PROGRAM MAIN
VAR
	fb_led_Show: FB_LedShow;
	btn_reset: BOOL;
	CPMU_PLC_Reset: PLC_Reset;
	d_state: DINT;
	CPMU_PLC_Start: PLC_Start;
	powerStatus:BOOL;

(*TwinSAFE*)
	Safe_run AT%Q*:BOOL;
	Err_Ack AT %Q*:BOOL;
	Estop_RunAndRestart AT %Q*:BOOL;
	AX5805_Error_Ack AT %Q*:BOOL;
	Led_Run  AT %Q*:BOOL;
	Led_Error  AT %Q*:BOOL;

	FB_ERROR AT%I*:BOOL;
	COM_ERROR AT%I*:BOOL;
	//OUT_ERROR AT%I*:BOOL;
	Estop_Out AT%I*:BOOL;

	SafeStatus:INT;
	SafePLCRunOK: BOOL;
	fb_ton: TON;
	fb_ton2: TON;
	fb_ton3: TON;
	fb_ton1: TON;
	fb_ton0: TON;
(*IO*)
	el1808_D1  AT%I* :ARRAY[1..4] OF BOOL;
	el1008 AT%I*:BOOL;
	EStopTrig:BOOL;
(*setAxisPosition*)
	SetAxisPosState: INT;
	FB_Set_AxisPosition:FB_SetAxisPosition;
	fb_ton4: TON;
	fb_ton5: TON;
	fb_ton6: TON;
	SetAxisPositionDone: BOOL;

	i: INT;
	j: INT;

(****RS232***)
	fbEL6001	: FB_SerialCom;
	
	moveDonePhaseShifter: BOOL;


(*Torque*)
	Torque_PS AT%I*:INT;
(**)
	btn_setAxisPosition: BOOL;
	ValueSet_PhaseShifterLin:LREAL;
(**)
	RestartTC: TC_Restart;
	
(*recipe*)
	RecipeINT:INT;
	RecipeBOOL:BOOL;
	RecipeManCommands: RecipeManCommands;
	SaveParameter : BOOL;  //保存文件
	LoadParameter : BOOL;  //读取文件
	Save_R_TRIG   : R_TRIG;
	Read_R_TRIG   : R_TRIG;
	loadparameterStatus: INT;
	RecipeBOOL2:BOOL;
	ReturnDwordLoad: DWORD;
	InsertionDeviceName:STRING;
(*UserMode*)
	pbUserMode: BOOL:=TRUE;
	EL1904 AT%I* :ARRAY[1..24] OF BOOL;
	setAxisPositionEnable: BOOL;
	state_loadParameters: INT;
	state_setLEPosBias: INT;
	//
	PositionBiasSet:BOOL;
	MC_SetLEPosBias_PhaseShifter:MC_WriteParameter;
	PositionBias_PhaseShifter: LREAL:=10.1;
	LoadLEPB_R_TRIG: R_TRIG;
	PositionBiasTON: TON;
	
	//
	OPC_TEST_Bi:BOOL:=TRUE; (*~ (OPC:1:available for OPC Clients) *)
	OPC_TEST_Bi2:BOOL;(*~ (OPC:1:available for OPC Clients) *)
	//
	HasTemperatureSensorOrNot:BOOL;//Only IVU or CPMU
	(*Sensor Reading*)
	Sensor_Reading_1 AT %I*:ARRAY[0..3] OF BYTE;
	Sensor_Reading_2 AT %I*:ARRAY[0..3] OF BYTE;
	Sensor_Reading_3 AT %I*:ARRAY[0..3] OF BYTE;
	Sensor_Reading_4 AT %I*:ARRAY[0..3] OF BYTE;
	Sensor_Reading_5 AT %I*:ARRAY[0..3] OF BYTE;
	Sensor_Reading_6 AT %I*:ARRAY[0..3] OF BYTE;
	Sensor_Reading_7 AT %I*:ARRAY[0..3] OF BYTE;
	Sensor_Reading_8 AT %I*:ARRAY[0..3] OF BYTE;
	Sensor_Reading_DpState AT %I*:USINT;
	Sensor_Reading_ExtDiagFlag AT %I*:BOOL;
	TemperatureSensors_1:LREAL;
	TemperatureSensors_2:LREAL;
	TemperatureSensors_3:LREAL;
	TemperatureSensors_4:LREAL;
	TemperatureSensors_5:LREAL;
	TemperatureSensors_6:LREAL;
	TemperatureSensors_7:LREAL;
	TemperatureSensors_8:LREAL;
	dut_sensor_datas_1:DUT_SENSOR_DATAS_1;
	dut_sensor_datas_2:DUT_SENSOR_DATAS_2;
	dut_sensor_datas_3:DUT_SENSOR_DATAS_3;
	dut_sensor_datas_4:DUT_SENSOR_DATAS_4;
	dut_sensor_datas_5:DUT_SENSOR_DATAS_5;
	dut_sensor_datas_6:DUT_SENSOR_DATAS_6;
	dut_sensor_datas_7:DUT_SENSOR_DATAS_7;
	dut_sensor_datas_8:DUT_SENSOR_DATAS_8;
	//
	temperature_gradient_2_To_1:LREAL;
	temperature_gradient_3_To_2:LREAL;
	temperature_gradient_5_To_4:LREAL;
	temperature_gradient_6_To_5:LREAL;
	temperature_gradient_max:LREAL;
	//
	temperature_average:LREAL;
	A_SetLinearEncoderPositionBias_Enable: BOOL;
	
		//
	temperatureStatus:INT;//0：有传感器度数错误；1:常温；2:低温；3:常温和低温中间态
	CryogenicTemperatureThreshold:LREAL:=80;//80K以下归划分为低温
	RoomTemperatureThreshold:LREAL:=293;//293K以上划分为常温
	//CPMU cryogenix ON/FF
	CryogenicCompensationOn:BOOL;
	CryogenicCompensationConditionsReady:BOOL;
	CryogenicCompensation_LeftTop:LREAL;
	CryogenicCompensation_RightTop:LREAL;
	CryogenicCompensation_LeftBottom:LREAL;
	CryogenicCompensation_RightBottom:LREAL;
	CryogenicCompensationDone: BOOL;
	
(**)
	bDriveDiagMessageAndNumber  : BOOL;
	m_GetDriveStatusState:INT;
	GetDriveStatusStateDone:BOOL;
	GetDriveStatusStateError:BOOL;
	GetDriveStatusTON: TON;
	//	
	fb_SoEReadDiagMessage_PhaseShifter: FB_SoEReadDiagMessage;
	DriveDiagMessage_PhaseShifter:STRING;
	//
	FB_SoEReadDiagNumber_PhaseShifter: FB_SoEReadDiagNumber;
	DriveDiagNumber_PhaseShifter:UDINT;
	bReloadDriveDiagMessageAndNumber: BOOL;
	
	(*load IOC*)
	bExe_load_Prog: BOOL;
	NT_StartProcess_Load: NT_StartProcess;
	Exe_load_step: UINT;
	R_TRIG_ExeLoad: R_TRIG;
	Exe_Load_Done:BOOL;
	(*kill IOC*)
	bExe_Kill_Prog: BOOL;
	NT_StartProcess_Kill: NT_StartProcess;
	Exe_kill_step: UINT;
	R_TRIG_Exekill: R_TRIG;
	Exe_Kill_Done:BOOL;

	KS_RightBottom_Near_Contact2: BOOL;
	
	//
	//more parameters get:gear;feedback2 direction 
	//
	//GetMoreDriveStatus_FunctionON:BOOL:=TRUE;
	GetDriveStatusTON2: TON;
	//GearNumerator,st182
	st_p182_PhaseShifter:ST_P182;
	FB_SoERead_GearNumerator_PhaseShifter: FB_SoERead;
	GearNumeratorGet_PhaseShifter:UDINT;
	GearNumeratorConfigured_PhaseShifter:UDINT;
	//GearDenominator,st183
	st_p183_PhaseShifter:ST_P183;
	FB_SoERead_GearDenominator_PhaseShifter: FB_SoERead;
	GearDenominatorGet_PhaseShifter:UDINT;
	GearDenominatorConfigured_PhaseShifter:UDINT;
	//Feedback2direction,st180
	st_p180_PhaseShifter:ST_P180;
	FB_SoERead_Feedback2direction_PhaseShifter: FB_SoERead;
	Feedback2directionGet_PhaseShifter:UINT;
	Feedback2directionConfigured_PhaseShifter:UINT;
	//
	//RestartDrivers
		(*重启驱动器*)
	btn_RestartDriversAll:BOOL;
	btn_RestartDriver1:BOOL;
	btn_RestartDriver2:BOOL;
	btn_RestartDriver3:BOOL;
	btn_RestartDriver4:BOOL;
	btn_RestartDriver5:BOOL;
	btn_RestartDriver6:BOOL;
	btn_RestartDriver7:BOOL;
	btn_RestartDriver8:BOOL;
	Relay_EL2624 AT %Q*:ARRAY[0..7]OF  BOOL;
	RestartDriver_RTRIG:R_TRIG;
	RestartDriver_TON:TON;
	RestartDriver_Triggered:BOOL;
	RestartDriver_State:DINT;
	RestartDriver_Done:BOOL;
	
	//
	//	LEHeartBeatMonitorFunction
	//
	LEHeartBeatMonitorFunctionOn: BOOL;
	LEHeartBeatFirstScan:BOOL;
	LEHeartBeatDeadZone : LREAL := 0; 
	LEHeartBeatAlarmTime : TIME := T#0.1S;
	
    //Pos_LeftTopLin_Last : LREAL; 
	Velo_PhaseShifterLin_Last : LREAL; 
	Pos_PhaseShifterMotor_Initial : LREAL; 
    StableTimer_PhaseShifterLin : TON; 
    StableTime_PhaseShifterLin : TIME; 
    DeltaVelo_PhaseShifterLin : LREAL; 
	IsInitialPositionSet_PhaseShifter: BOOL;
	MotorPosChange_PhaseShifter: LREAL;
	Threshold_PhaseShifterMotorPos:LREAL:=0.1;
	Threshold_PhaseShifterMotorVelo:LREAL:=0.2;
	Alarm_PhaseShifterLin:BOOL;
	Alarm_PhaseShifterMotorPos:BOOL;
	Alarm_PhaseShifterMotorVelo:BOOL;
	
	(*setAxisPosition*)
	SetMotorAxisPosState: INT;
	FB_Set_MotorAxisPosition:FB_SetMotorAxisPosition;
	fb_ton4_2: TON;
	fb_ton5_2: TON;
	fb_ton6_2: TON;
	SetMotorAxisPositionDone: BOOL;
	
	btn_SetMotorAxisPosition: BOOL;
	MonitorMotorAndLEFunctionOn:BOOL:=TRUE;
	
	(*GetMotorTempture*)
	MotorTemperature AT %I*:ARRAY[0..1] OF UINT;
	MotorTemperature_PS:LREAL;
END_VAR

(*MaintenanceMode*)
IF MaintenanceMode THEN
	MaintenanceModeLed:=TRUE;
	RETURN;
ELSE
	MaintenanceModeLed:=FALSE;	
END_IF

(*加载Ricipe参数*)
A_InitRecipeParameters();
(*Restart TwinCAT*)
IF Global_Variables.m_restartTC THEN
(*首先关闭opcIocShell.exe*)	
	bExe_Kill_Prog:=TRUE;
	A_KillOpcIocShellExe();
(*重启TC*)
	IF Exe_Kill_Done THEN
		A_RestartTC();
	END_IF
END_IF
(*******InitAxisParameters*******)
A_InitAxisParameters();
(*******CheckLimitSwitch*******)
A_CheckLimitSwitch();
(*Check Kill Switch*)
A_CheckKillSwitch();
(*******PosDiff¼à¿Ø*******)
A_PosDiffDetectiion();
(*******³õÊ¼»¯SafePlc*******)
IF NOT simulation THEN
A_SafePlcStartInit();
END_IF
(************SetAxisPosition*********************)
IF  NOT USELinearEncoder AND setAxisPositionEnable AND btn_setAxisPosition THEN
	//IF NOT SerAxisPositionDone THEN
		FB_Set_AxisPosition.ValueSet_PhaseShifterLin:=ValueSet_PhaseShifterLin;
		A_SetAxisPosition();
	//END_IF
END_IF
(*******³Mode Select******)
IF SafePLCRunOK OR Simulation THEN
	UserMode();
END_IF
(*******Led Show******)
fb_led_Show();
(*******Check Power status******)
FB_Power(Check:=TRUE);
st_Power:=FB_Power.PowerState;
(*********RS232*********************)
BackgroundEL();
(*fbEL6001(TxBuffer:=TxBufferEL, RxBuffer:=RxBufferEL);*)

(*设置position bias*)
IF loadParametersDone AND (DriveStatus=1 OR simulation) THEN 
	A_SetLinearEncoderPositionBias();
END_IF
(*检查硬急停状态，包括安全限位、柜门急停、手持急停*)
A_CheckHardwareEmergencyStopStatus();
(*获取驱动器状态信息*)
IF NOT simulation THEN
	A_GetDriverStatus();
END_IF
(*IDControlReady*)
IF ((DriveStatus<>0 AND SafePLCRunOK) OR simulation) AND NOT Error THEN
	IDControlReady:=TRUE;
ELSE
	IDControlReady:=FALSE;
END_IF

(*IOC Start*)
//IF IDControlReady THEN
	bExe_load_Prog:=TRUE;
	A_LoadOpcIocShellExe();
//END_IF

(*检查光栅读数是否在范围内*)
A_CheckLinearEncoder();

(*RestartDrivers*)
A_RestartDrivers();

(*A_LEHeartBeatMonitor*)
IF LEHeartBeatMonitorFunctionOn THEN
	A_LEHeartBeatMonitor();
END_IF
(************SetMotorAxisPosition*********************)
//IDControl 1s after
fb_ton5_2.IN:=IDControlReady;
fb_ton5_2.PT:=T#1S;
fb_ton5_2();
IF fb_ton5_2.Q THEN
	btn_SetMotorAxisPosition:=TRUE;
END_IF
IF  USELinearEncoder AND btn_SetMotorAxisPosition THEN
	IF NOT SetMotorAxisPositionDone THEN
		FB_Set_MotorAxisPosition.ValueSet_PhaseShifterMotor:=Pos_PhaseShifterLin;
		A_SetMotorAxisPosition();
	END_IF
END_IF
(*A_MonitorMotorAndLE*)
IF MonitorMotorAndLEFunctionOn AND SetMotorAxisPositionDone THEN
	A_MonitorMotorAndLE();
END_IF
(*A_CheckMaxVelocity*)
A_CheckMaxVelocity();

ACTION A_CheckHardwareEmergencyStopStatus:
IF 	NOT KS_TopNear_Contact1 OR
	NOT KS_TopNear_Contact2 OR
	NOT KS_TopFar_Contact1 OR
	NOT KS_TopFar_Contact2 OR
	
(*E-STOP*)
	NOT KS_CabinetEmergency_contact1 OR
	NOT KS_CabinetEmergency_contact2 OR
	NOT KS_handEmergency1_Contact1 OR
	NOT KS_handEmergency1_Contact2 OR
	NOT KS_handEmergency2_Contact1 OR
	NOT KS_handEmergency2_Contact2 OR
	NOT KS_softEmergency2_Contact THEN
	Hardware_EmergencyStop:=FALSE;
ELSE
	Hardware_EmergencyStop:=TRUE;
END_IF
END_ACTION

ACTION A_CheckKillSwitch:
IF simulation THEN	
	KS_TopFar_Contact1:=TRUE;	
	KS_TopFar_Contact2:=TRUE;	
	KS_TopNear_Contact1:=TRUE;	
	KS_TopNear_Contact2:=TRUE;	
	KS_BottomFar_Contact1:=TRUE;	
	KS_BottomFar_Contact2:=TRUE;	
	KS_BottomNear_Contact1:=TRUE;	
	KS_BottomNear_Contact2:=TRUE;	
	(*E-STOP*)
	KS_CabinetEmergency_contact1:=TRUE;
	KS_CabinetEmergency_contact2:=TRUE;	
	KS_handEmergency1_Contact1:=TRUE;
	KS_handEmergency1_Contact2:=TRUE;
	KS_handEmergency2_Contact1:=TRUE;
	KS_handEmergency2_Contact2:=TRUE;
	
	KS_softEmergency2_Contact:=TRUE;

ELSE
	KS_TopFar_Contact1:=EL1904[1];//c1	
	KS_TopFar_Contact2:=EL1904[2];//c1	
	KS_TopNear_Contact1:=EL1904[3];//c1	
	KS_TopNear_Contact2:=EL1904[4];//c1	
	KS_BottomFar_Contact1:=EL1904[5];//c2	
	KS_BottomFar_Contact2:=EL1904[6];//c2	
	KS_BottomNear_Contact1:=EL1904[7];//c2	
	KS_BottomNear_Contact2:=EL1904[8];//c2
	
	
	(*E-STOP*)
	KS_CabinetEmergency_contact1:=EL1904[9];//c3
	KS_CabinetEmergency_contact2:=EL1904[10];//c3
	
	KS_handEmergency1_Contact1:=EL1904[11];//c3
	KS_handEmergency1_Contact2:=EL1904[12];//c3
	KS_handEmergency2_Contact1:=EL1904[13];//c4
	KS_handEmergency2_Contact2:=EL1904[14];//c4
	
	KS_softEmergency2_Contact:=EL1904[15];//c4
	//c4
	END_IF
END_ACTION

ACTION A_CheckLimitSwitch:
(*******1.´ÓIO»ñÈ¡ÏÞÎ»×´Ì¬******)
(**)
IF simulation THEN
	(**)
	LS_TopFar  :=TRUE;
	LS_TopNear :=TRUE;
	LS_BottomFar :=TRUE;
	LS_BottomNear  :=TRUE;
ELSE
	LS_TopFar  :=el1808_D1[1];
	LS_TopNear :=el1808_D1[2];
	LS_BottomFar :=el1808_D1[3];
	LS_BottomNear :=el1808_D1[4];

END_IF
(******2.TopÏÞÎ»»òÕßBottomÏÞÎ»ÓÐÒ»¸ö´¥·¢£¬È«¾Ö±äÁ¿¡£¸øMC_POWERÓÃÓÚ·½Ïò¿ØÖÆ£¬ÓÐÒ»¸öÏÞÎ»Îª´¥·¢ÎªFALSE£¬ÔòUnreach_LSÎªFALSE******)
//Unreach_LS_Far:=LS_TopFar AND LS_BottomFar;
//Unreach_LS_Near:=LS_TopNear AND LS_BottomNear;

Unreach_LS_Far:=LS_TopFar;
Unreach_LS_Near:=LS_TopNear;
END_ACTION

ACTION A_CheckLinearEncoder:
//LEProtectionPosition
min_UserLEProtectionGapPosition:=min_UserGapPositionNew-min_ThresholdGapSoft2LEProtection;//回程误差有0.1mm
max_UserLEProtectionGapPosition:=max_UserGapPositionNew+max_ThresholdGapSoft2LEProtection;

//如果没有使用光栅、或者光栅参数没设置好，则不检查光栅位置
IF NOT USELinearEncoder OR NOT PositionBiasDone THEN
	RETURN;
END_IF
IF Pos_PhaseShifterLin <=0 THEN
	ErrorID:=1101;
	Error:=TRUE;
	ErrorDescription:='Pos_PhaseShifterLin <=0';
	FB_PlcEmergencyStop();
	LED_Error:=TRUE;
END_IF
//

IF Pos_PhaseShifterLin >max_UserLEProtectionGapPosition THEN
	ErrorID:=1105;
	Error:=TRUE;
	ErrorDescription:='Pos_PhaseShifterLin >max_UserLEProtectionGapPosition';
	FB_PlcEmergencyStop();
	LED_Error:=TRUE;
END_IF

//
IF Pos_PhaseShifterLin <min_UserLEProtectionGapPosition THEN
	ErrorID:=1109;
	Error:=TRUE;
	ErrorDescription:='Pos_PhaseShifterLin <min_UserLEProtectionGapPosition';
	FB_PlcEmergencyStop();
	LED_Error:=TRUE;
END_IF
END_ACTION

ACTION A_CheckMaxVelocity:
IF NOT USELinearEncoder OR NOT PositionBiasDone OR NOT IDControlReady THEN
	RETURN;
END_IF
IF NOT st_Power THEN
	RETURN;
END_IF
//Monitoring Motor and LE Position/Velocity
MaxVelocityGlobalVelocity:=MAX(max_UserGapVelocityNew,max_UserTaperVelocityNew,UserMode.max_SS_StepVelocity,
			UserMode.Global_ChainProtection_MPS_MoveVelocity,UserMode.Global_ChainProtection_EPS_MoveVelocity);
IF 	ABS(Velo_PhaseShifterLin) > MaxVelocityGlobalVelocity*1.1/2 THEN
	ErrorID:=7001;
	Error:=TRUE;
	ErrorDescription:='ABS(Velo_PhaseShifterLin) > MaxVelocityGlobalVelocity*1.1/2';
	FB_PlcEmergencyStop();
	LED_Error:=TRUE;
END_IF
IF 	ABS(Velo_PhaseShifterMotor) > MaxVelocityGlobalVelocity*1.1/2 THEN
	ErrorID:=7002;
	Error:=TRUE;
	ErrorDescription:='ABS(Velo_PhaseShifterMotor) > MaxVelocityGlobalVelocity*1.1/2';
	FB_PlcEmergencyStop();
	LED_Error:=TRUE;
END_IF
END_ACTION

ACTION A_GetDriverStatus:
//
//DriveMessage/Drive Number/Gear number/feedback2 direction
//
IF bReloadDriveDiagMessageAndNumber THEN
	m_GetDriveStatusState:=0;
	bReloadDriveDiagMessageAndNumber:=FALSE;
END_IF
GetDriveStatusTON(PT:=T#1S);
GetDriveStatusTON2(PT:=T#0.1S);
A_GetDriverStatusMC();
CASE m_GetDriveStatusState OF
	0:
		GetDriveStatusTON.IN:=TRUE;
		m_GetDriveStatusState:=1;
	1:
		IF GetDriveStatusTON.Q THEN
			bDriveDiagMessageAndNumber:=TRUE;
			m_GetDriveStatusState:=2;
		END_IF
	2:
		GetDriveStatusTON.IN:=FALSE;
		DriveDiagMessage_PhaseShifter:=fb_SoEReadDiagMessage_PhaseShifter.sDiagMessage.strData;
		//
		DriveDiagNumber_PhaseShifter:=FB_SoEReadDiagNumber_PhaseShifter.iDiagNumber;
		//
		GearNumeratorGet_PhaseShifter:=st_p182_PhaseShifter.Feedback_2_geat_numerator;
		//
		GearDenominatorGet_PhaseShifter:=st_p183_PhaseShifter.Feedback_2_geat_denominator;
		//
		Feedback2directionGet_PhaseShifter:=st_p180_PhaseShifter.Feedback_direction;
		//
		IF 	NOT fb_SoEReadDiagMessage_PhaseShifter.bBusy
			AND NOT FB_SoEReadDiagNumber_PhaseShifter.bBusy
			AND NOT FB_SoERead_GearNumerator_PhaseShifter.bBusy 
			AND NOT FB_SoERead_GearDenominator_PhaseShifter.bBusy 
			AND NOT FB_SoERead_Feedback2direction_PhaseShifter.bBusy  THEN
				GetDriveStatusTON2.IN:=TRUE;
				IF GetDriveStatusTON2.Q THEN
					m_GetDriveStatusState:=88;
				END_IF
		END_IF
		IF 	fb_SoEReadDiagMessage_PhaseShifter.bError
			OR FB_SoEReadDiagNumber_PhaseShifter.bError
			OR FB_SoERead_GearNumerator_PhaseShifter.bError 
			OR FB_SoERead_GearDenominator_PhaseShifter.bError 
			OR FB_SoERead_Feedback2direction_PhaseShifter.bError 
		THEN
			m_GetDriveStatusState:=-100;
		END_IF
		
	88:
		bDriveDiagMessageAndNumber:=FALSE;
		A_GetDriverStatusMC();
		GetDriveStatusStateDone:=TRUE;
		GetDriveStatusStateError:=FALSE;
		//
		(*Drive Status*)
		//D012, Axis state machine: Control and power section ready,53266
		IF DriveDiagNumber_PhaseShifter=16#D012  THEN
			DriveStatus:=1;
		//D013, Axis state machine: Axis in operation,53267
		ELSIF DriveDiagNumber_PhaseShifter=16#D013  THEN
			DriveStatus:=2;
		//D014，Axis state machine: Axis halt.53266和53267中间会经历这么一个状态，算正常状态
		ELSIF DriveDiagNumber_PhaseShifter=16#D014  THEN
			DriveStatus:=3;
		ELSE
			DriveStatus:=0;
		END_IF
		//
		//
		//	//check statusGet and status configured
		IF 	GearNumeratorGet_PhaseShifter<>GearNumeratorConfigured_PhaseShifter 
			OR GearDenominatorGet_PhaseShifter<>GearDenominatorConfigured_PhaseShifter   THEN
				bDriveDiagMessageAndNumber:=FALSE;
				A_GetDriverStatusMC();
				GetDriveStatusStateDone:=FALSE;
				GetDriveStatusStateError:=TRUE;
				Error:=TRUE;
				ErrorId:=1302;
				ErrorDescription:='gearParameters Error';
				Plc_EmergencyStop:=FALSE;
		END_IF
		IF USELinearEncoder THEN
			IF  Feedback2directionGet_PhaseShifter<>Feedback2directionConfigured_PhaseShifter THEN
					bDriveDiagMessageAndNumber:=FALSE;
					A_GetDriverStatusMC();
					GetDriveStatusStateDone:=FALSE;
					GetDriveStatusStateError:=TRUE;
					Error:=TRUE;
					ErrorId:=1303;
					ErrorDescription:='fb2direction Error';
					Plc_EmergencyStop:=FALSE;
			END_IF
		END_IF
		m_GetDriveStatusState:=0;
	-100:
		bDriveDiagMessageAndNumber:=FALSE;
		A_GetDriverStatusMC();
		GetDriveStatusStateDone:=FALSE;
		GetDriveStatusStateError:=TRUE;
		Error:=TRUE;
		ErrorId:=1301;
		ErrorDescription:='GetDriveStatusStateError';
END_CASE
END_ACTION

ACTION A_GetDriverStatusMC:
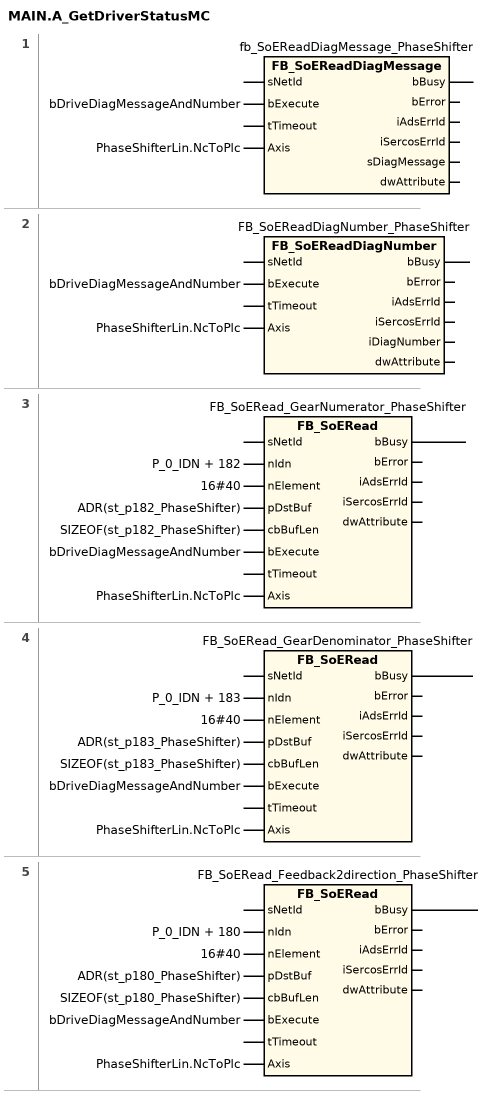
// NETWORK 1
fb_SoEReadDiagMessage_PhaseShifter(bExecute := bDriveDiagMessageAndNumber, Axis := PhaseShifterLin.NcToPlc); // FB_SoEReadDiagMessage

// NETWORK 2
FB_SoEReadDiagNumber_PhaseShifter(bExecute := bDriveDiagMessageAndNumber, Axis := PhaseShifterLin.NcToPlc); // FB_SoEReadDiagNumber

// NETWORK 3
FB_SoERead_GearNumerator_PhaseShifter(
    nIdn := P_0_IDN + 182,
    nElement := 16#40,
    pDstBuf := ADR(st_p182_PhaseShifter),
    cbBufLen := SIZEOF(st_p182_PhaseShifter),
    bExecute := bDriveDiagMessageAndNumber,
    Axis := PhaseShifterLin.NcToPlc); // FB_SoERead

// NETWORK 4
FB_SoERead_GearDenominator_PhaseShifter(
    nIdn := P_0_IDN + 183,
    nElement := 16#40,
    pDstBuf := ADR(st_p183_PhaseShifter),
    cbBufLen := SIZEOF(st_p183_PhaseShifter),
    bExecute := bDriveDiagMessageAndNumber,
    Axis := PhaseShifterLin.NcToPlc); // FB_SoERead

// NETWORK 5
FB_SoERead_Feedback2direction_PhaseShifter(
    nIdn := P_0_IDN + 180,
    nElement := 16#40,
    pDstBuf := ADR(st_p180_PhaseShifter),
    cbBufLen := SIZEOF(st_p180_PhaseShifter),
    bExecute := bDriveDiagMessageAndNumber,
    Axis := PhaseShifterLin.NcToPlc); // FB_SoERead
END_ACTION

ACTION A_GetMotorTemperature:
MotorTemperature_PS:=UINT_TO_LREAL(MotorTemperature[0])/10;
END_ACTION

ACTION A_InitAxisParameters:
//LE	
	Pos_PhaseShifterLin:=DINT_TO_LREAL(LREAL_TO_DINT(PhaseShifterLin.NcToPlc.ActPos*100000))/100000;
	moveStatusPhaseShifterLin:=PhaseShifterLin.Status.Moving;
	Velo_PhaseShifterLin:=DINT_TO_LREAL(LREAL_TO_DINT(PhaseShifterLin.NcToPlc.ActVelo*100000))/100000;
	PosDiff_PhaseShifterLin_actual:=DINT_TO_LREAL(LREAL_TO_DINT(PhaseShifterLin.NcToPlc.PosDiff*100000))/100000;
	Torque_PhaseShifterLin:=PhaseShifterLin.NcToPlc.ActTorque;	
	PhaseShifterLin.ReadStatus();

//Motor
	Pos_PhaseShifterMotor:=DINT_TO_LREAL(LREAL_TO_DINT(PhaseShifterMotor.NcToPlc.ActPos*100000))/100000;
	moveStatusPhaseShifterMotor:=PhaseShifterMotor.Status.Moving;
	Velo_PhaseShifterMotor:=DINT_TO_LREAL(LREAL_TO_DINT(PhaseShifterMotor.NcToPlc.ActVelo*100000))/100000;
	PosDiff_PhaseShifterMotor_actual:=DINT_TO_LREAL(LREAL_TO_DINT(PhaseShifterMotor.NcToPlc.PosDiff*100000))/100000;
	Torque_PhaseShifterMotor:=PhaseShifterMotor.NcToPlc.ActTorque;	
	PhaseShifterMotor.ReadStatus();

//
	//get Delta
	//
	//Delta Pos
	DeltaPos_PhaseShifter:=Pos_PhaseShifterLin - Pos_PhaseShifterMotor;
	//Delta Velocity	
	DeltaVelo_PhaseShifter:=Velo_PhaseShifterLin - Velo_PhaseShifterMotor;
	//Delta lagDistance
	DeltaPosDiff_PhaseShifter_actual:=PosDiff_PhaseShifterLin_actual - PosDiff_PhaseShifterMotor_actual;
	//Delta Torque
	DeltaTorque_PhaseShifter:=Torque_PhaseShifterLin - Torque_PhaseShifterMotor;
END_ACTION

ACTION A_InitRecipeParameters:
CASE state_loadParameters OF
	0:
		LoadParameter:=TRUE;
		Read_R_TRIG(CLK:=LoadParameter , Q=> );
		IF Read_R_TRIG.Q THEN
			state_loadParameters:=1;
		END_IF
	1:
		 ReturnDwordLoad:=RecipeManCommands.LoadAndWriteRecipe(RecipeDefinitionName:='Recipes' , RecipeName:='ParametersPS');
    	 LoadParameter:=FALSE;
		 IF ReturnDwordLoad<>0 THEN
		 	state_loadParameters:=-100;
		ELSE
			LoadRecipeParameters:=TRUE;
			LoadParameter:=FALSE;
			state_loadParameters:=88;
	 	END_IF
	88:
		loadParametersDone:=TRUE;
	-100:
		loadParametersDone:=FALSE;
		Error:=TRUE;
		ErrorId:=101;
		ErrorDescription:='LoadRecipeParameters Error';
		Plc_EmergencyStop:=FALSE;
END_CASE
//Save_R_TRIG(CLK:=SaveParameter , Q=> );
Read_R_TRIG(CLK:=LoadParameter , Q=> );
//IF Save_R_TRIG.Q THEN  //将plc数据以文件形式保存在工控机中
//	 RecipeManCommands.CreateRecipe(RecipeDefinitionName:='Recipes' , RecipeName:='ParametersPS2' );
//	 RecipeManCommands.ReadAndSaveRecipe(RecipeDefinitionName:='Recipes' , RecipeName:='ParametersPS2' );
//	 SaveParameter:=FALSE;
//END_IF
IF Read_R_TRIG.Q THEN  //将工控机中的文件数据读取到plc中
     ReturnDwordLoad:=RecipeManCommands.LoadAndWriteRecipe(RecipeDefinitionName:='Recipes' , RecipeName:='ParametersPS');
     LoadParameter:=FALSE;
	 IF ReturnDwordLoad<>0 THEN
		 Error:=TRUE;
		 ErrorId:=101;
		 ErrorDescription:='LoadRecipeParameters Error';
		 Plc_EmergencyStop:=FALSE;
	 END_IF
END_IF
END_ACTION

ACTION A_KillOpcIocShellExe:
R_TRIG_Exekill(CLK:=bExe_Kill_Prog, Q=> );
CASE Exe_kill_step OF
	0:
		IF R_TRIG_Exekill.Q THEN
			NT_StartProcess_Kill.START:=FALSE;
			NT_StartProcess_Kill.PATHSTR:='C:\HZB\OpcIocShell\IDControlIOC\killcmd.bat';
			//NT_StartProcess_Kill.DIRNAME:='C:\Program Files (x86)\HZB\OpcIocShell\bin\opcIocShell.exe';
			Exe_kill_step:=10;
		END_IF;
	10:
		NT_StartProcess_Kill.START:=TRUE;
		Exe_kill_step:=20;
	20:
		IF NT_StartProcess_Kill.ERR THEN
			Exe_kill_step:=0;
		ELSE
			Exe_kill_step:=30;
		END_IF;

	30:
		NT_StartProcess_Kill.START:=TRUE;
		Exe_kill_step:=40;
	40:
		IF NOT NT_StartProcess_Kill.BUSY THEN
			NT_StartProcess_Kill.START:=FALSE;
			Exe_Kill_Done:=TRUE;
			Exe_kill_step:=0;
		END_IF;
END_CASE;

NT_StartProcess_Kill(
	NETID:='' ,
	PATHSTR:= ,
	DIRNAME:= , 
	COMNDLINE:= , 
	START:= ,
	ERRID=> );
END_ACTION

ACTION A_LEHeartBeatMonitor:
//monitor only while power on and not simulation or not use LE
IF NOT st_Power THEN
	RETURN;
END_IF
(**)
IF simulation THEN
	RETURN;
END_IF
IF NOT USELinearEncoder THEN
	RETURN;
END_IF

// 初始化
IF LEHeartBeatFirstScan THEN
    Velo_PhaseShifterLin_Last := PhaseShifterLin.NcToPlc.ActVelo;
    LEHeartBeatFirstScan := FALSE;
END_IF;

// 计算光栅前后速度差，速度差比位置差更敏感
DeltaVelo_PhaseShifterLin := ABS(PhaseShifterLin.NcToPlc.ActVelo - Velo_PhaseShifterLin_Last);
//PhaseShifter monitor
IF DeltaVelo_PhaseShifterLin > LEHeartBeatDeadZone THEN
    // 有变动，光栅正常，计数器归零，更新位置,重置所有状态
    StableTimer_PhaseShifterLin(IN := FALSE, PT := LEHeartBeatAlarmTime);
    Alarm_PhaseShifterLin := FALSE;
    Velo_PhaseShifterLin_Last := PhaseShifterLin.NcToPlc.ActVelo;  // 
    StableTime_PhaseShifterLin := T#0S;
	IsInitialPositionSet_PhaseShifter:=FALSE;
	Alarm_PhaseShifterMotorPos:=FALSE;
	Alarm_PhaseShifterMotorVelo:=FALSE;
ELSE
    //一点变动没有了，光栅异常，开始计时
    StableTimer_PhaseShifterLin(
        IN := TRUE,
        PT := LEHeartBeatAlarmTime,
        ET => StableTime_PhaseShifterLin
    );
	//记录电机初始位置，后后续对比做准备
	IF NOT IsInitialPositionSet_PhaseShifter THEN
        Pos_PhaseShifterMotor_Initial := Pos_PhaseShifterMotor;  // 记录初始位置
        IsInitialPositionSet_PhaseShifter := TRUE;
   	END_IF;
    
    // 100ms速度完全不变，开始监控电机速度和位置
    IF StableTimer_PhaseShifterLin.Q THEN
        Alarm_PhaseShifterLin := TRUE;  // 
			//电机位置对比及监测
			MotorPosChange_PhaseShifter:=ABS( Pos_PhaseShifterMotor-Pos_PhaseShifterMotor_Initial);
			IF MotorPosChange_PhaseShifter > Threshold_PhaseShifterMotorPos THEN
				Alarm_PhaseShifterMotorPos:=TRUE;
				ErrorID:=5001;
				ErrorDescription:='5001';
				Error:=TRUE;
				FB_PlcEmergencyStop();
				LED_Error:=TRUE;
			ELSE
				Alarm_PhaseShifterMotorPos:=FALSE;
			END_IF
			//电机速度监测
			IF Velo_PhaseShifterMotor > Threshold_PhaseShifterMotorVelo THEN
				Alarm_PhaseShifterMotorVelo:=TRUE;
				ErrorID:=5002;
				ErrorDescription:='5002';
				Error:=TRUE;
				FB_PlcEmergencyStop();
				LED_Error:=TRUE;
			ELSE
				Alarm_PhaseShifterMotorVelo:=FALSE;
			END_IF
    ELSE
        Alarm_PhaseShifterLin := FALSE;
	END_IF
END_IF
END_ACTION

ACTION A_LoadOpcIocShellExe:
R_TRIG_Exeload(CLK:=bExe_load_Prog, Q=> );
CASE Exe_load_step OF
	0:
		IF R_TRIG_Exeload.Q THEN
			NT_StartProcess_Load.START:=FALSE;
			NT_StartProcess_Load.PATHSTR:='C:\HZB\OpcIocShell\IDControlIOC\startTwinCATOPCServer.bat';
			Exe_load_step:=10;
		END_IF;
	10:
		NT_StartProcess_Load.START:=TRUE;
		Exe_load_step:=20;
	20:
		IF NT_StartProcess_Load.ERR THEN
			Exe_load_step:=0;
		ELSE
			Exe_load_step:=30;
		END_IF;
	30:
		IF NOT NT_StartProcess_Load.BUSY THEN
			NT_StartProcess_Load.START:=FALSE;
			Exe_Load_Done:=TRUE;
			Exe_load_step:=0;
		END_IF;
END_CASE;

NT_StartProcess_Load(
	NETID:='' ,
	PATHSTR:= ,
	DIRNAME:= , 
	COMNDLINE:= , 
	START:= ,
	ERRID=> );
END_ACTION

ACTION A_MonitorMotorAndLE:
//Monitoring Motor and LE Position/Velocity
IF 	ABS(DeltaPos_PhaseShifter) > ThresholdDeltaPos_PhaseShifter THEN
	ErrorID:=6001;
	Error:=TRUE;
	ErrorDescription:='ABS(DeltaPos_PhaseShifter) > ThresholdDeltaPos_PhaseShifter';
	FB_PlcEmergencyStop();
	LED_Error:=TRUE;
END_IF

IF ABS(DeltaVelo_PhaseShifter) > ThresholdDeltaVelo_PhaseShifter THEN
	ErrorID:=6002;
	Error:=TRUE;
	ErrorDescription:='ABS(DeltaVelo_PhaseShifter) > ThresholdDeltaVelo_PhaseShifter';
	FB_PlcEmergencyStop();
	LED_Error:=TRUE;
END_IF


(*
//
//IF NotMoving ,Threshold is less
//
IF NOT moveStatusLeftTop THEN
		IF 	ABS(DeltaPos_LeftTop) > ThresholdDeltaPos_LeftTop/3 THEN
		ErrorID:=6009;
		Error:=TRUE;
		ErrorDescription:='ABS(DeltaPos_LeftTop) > ThresholdDeltaPos_LeftTop/3';
		FB_PlcEmergencyStop();
		LED_Error:=TRUE;
	END_IF
END_IF
IF NOT moveStatusRightTop THEN
	IF ABS(DeltaPos_RightTop) > ThresholdDeltaPos_RightTop/3 THEN
		ErrorID:=6010;
		Error:=TRUE;
		ErrorDescription:='ABS(DeltaPos_RightTop) > ThresholdDeltaPos_RightTop/3';
		FB_PlcEmergencyStop();
		LED_Error:=TRUE;
	END_IF
END_IF
IF NOT moveStatusLeftBottom THEN
	IF ABS(DeltaPos_LeftBottom) > ThresholdDeltaPos_LeftBottom/3 THEN
		ErrorID:=6011;
		Error:=TRUE;
		ErrorDescription:='ABS(DeltaPos_LeftBottom) > ThresholdDeltaPos_LeftBottom/3';
		FB_PlcEmergencyStop();
		LED_Error:=TRUE;
	END_IF
END_IF
IF NOT moveStatusRightBottom THEN
	IF ABS(DeltaPos_RightBottom) > ThresholdDeltaPos_RightBottom/3 THEN
		ErrorID:=6012;
		Error:=TRUE;
		ErrorDescription:='ABS(DeltaPos_RightBottom) > ThresholdDeltaPos_RightBottom';
		FB_PlcEmergencyStop();
		LED_Error:=TRUE;
	END_IF
END_IF

//
IF NOT moveStatusLeftTop THEN
	IF ABS(DeltaVelo_LeftTop) > ThresholdDeltaVelo_LeftTop/3 THEN
		ErrorID:=6013;
		Error:=TRUE;
		ErrorDescription:='ABS(DeltaVelo_LeftTop) > ThresholdDeltaVelo_LeftTop/3';
		FB_PlcEmergencyStop();
		LED_Error:=TRUE;
	END_IF
END_IF
IF NOT moveStatusRightTop THEN
	IF ABS(DeltaVelo_RightTop) > ThresholdDeltaVelo_RightTop/3 THEN
		ErrorID:=6014;
		Error:=TRUE;
		ErrorDescription:='ABS(DeltaVelo_RightTop) > ThresholdDeltaVelo_RightTop/3';
		FB_PlcEmergencyStop();
		LED_Error:=TRUE;
	END_IF
END_IF
IF NOT moveStatusLeftBottom THEN
	IF ABS(DeltaVelo_LeftBottom) > ThresholdDeltaVelo_LeftBottom/3 THEN
		ErrorID:=6015;
		Error:=TRUE;
		ErrorDescription:='ABS(DeltaVelo_LeftBottom) > ThresholdDeltaVelo_LeftBottom/3';
		FB_PlcEmergencyStop();
		LED_Error:=TRUE;
	END_IF
END_IF
IF NOT moveStatusRightBottom THEN
	IF ABS(DeltaVelo_RightBottom) > ThresholdDeltaVelo_RightBottom/3 THEN
		ErrorID:=6016;
		Error:=TRUE;
		ErrorDescription:='ABS(DeltaVelo_RightBottom) > ThresholdDeltaVelo_RightBottom/3';
		FB_PlcEmergencyStop();
		LED_Error:=TRUE;
	END_IF
END_IF
*)
END_ACTION

ACTION A_PosDiffDetectiion:
IF ABS(PosDiff_PhaseShifterLin_actual)>PosDiff_PhaseShifterLin THEN
	ErrorID:=201;
	Error:=TRUE;
	ErrorDescription:='ABS(PosDiff_PhaseShifterLin_actual)>PosDiff_PhaseShifterLin';
	FB_PlcEmergencyStop();
	LED_Error:=TRUE;
END_IF
END_ACTION

ACTION A_RestartDrivers:
Relay_EL2624[0]:=btn_RestartDriver1;
Relay_EL2624[1]:=btn_RestartDriver2;
Relay_EL2624[2]:=btn_RestartDriver3;
Relay_EL2624[3]:=btn_RestartDriver4;
Relay_EL2624[4]:=btn_RestartDriver5;
Relay_EL2624[5]:=btn_RestartDriver6;
Relay_EL2624[6]:=btn_RestartDriver7;
Relay_EL2624[7]:=btn_RestartDriver8;
///
//1.上升沿触发，btn_RestartDrivers上升沿后，btn_RestartDriver1~8全部高电平
//2、3s后，Driver1~8全部恢复低电平
//3、恢复全部状态到初始
///
RestartDriver_RTRIG(CLK:=btn_RestartDriversAll);
IF RestartDriver_RTRIG.Q THEN
	RestartDriver_Triggered:=TRUE;
	RestartDriver_Done:=FALSE;
END_IF
IF RestartDriver_Triggered THEN
	CASE RestartDriver_State OF
		0:
			btn_RestartDriver1:=TRUE;
			btn_RestartDriver2:=TRUE;
			btn_RestartDriver3:=TRUE;
			btn_RestartDriver4:=TRUE;
			btn_RestartDriver5:=TRUE;
			btn_RestartDriver6:=TRUE;
			btn_RestartDriver7:=TRUE;
			btn_RestartDriver8:=TRUE;
			//计时开始
			RestartDriver_TON(PT:=T#10S);
			RestartDriver_TON.IN:=TRUE;
			IF RestartDriver_TON.Q THEN
				RestartDriver_State:=1;
			END_IF
		1:
			btn_RestartDriver1:=FALSE;
			btn_RestartDriver2:=FALSE;
			btn_RestartDriver3:=FALSE;
			btn_RestartDriver4:=FALSE;
			btn_RestartDriver5:=FALSE;
			btn_RestartDriver6:=FALSE;
			btn_RestartDriver7:=FALSE;
			btn_RestartDriver8:=FALSE;
			RestartDriver_State:=88;
		88:
			RestartDriver_TON.IN:=FALSE;
			btn_RestartDriversAll:=FALSE;
			RestartDriver_State:=0;
			RestartDriver_Triggered:=FALSE;
			RestartDriver_Done:=TRUE;
	END_CASE
END_IF
END_ACTION

ACTION A_RestartTC:
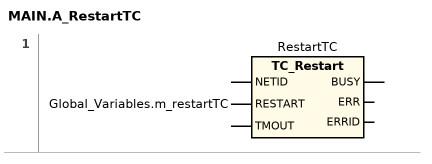
// NETWORK 1
RestartTC(RESTART := Global_Variables.m_restartTC); // TC_Restart
END_ACTION

ACTION A_SafePlcStartInit:
fb_ton0(PT:=t#1s);
fb_ton1(PT:=t#0.1s);
fb_ton2(PT:=t#0.1s);
fb_ton3(PT:=t#0.1s);

CASE SafeStatus OF
	0:
		IF COM_ERROR OR NOT Estop_Out THEN
			Err_Ack:=TRUE;
			fb_ton0.IN:=TRUE;
			SafeStatus:=1;
		ELSE
			SafePLCRunOK:=TRUE;
			SafeStatus:=0;
		END_IF
	1:
		IF fb_ton0.Q THEN
			Err_Ack:=FALSE;
			Safe_run:=TRUE;
			fb_ton1.IN:=TRUE;
			SafeStatus:=2;
		END_IF

	2:
		IF fb_ton1.Q THEN
			IF Estop_RunAndRestart=FALSE THEN
				Estop_RunAndRestart:=TRUE;
				fb_ton2.IN:=TRUE;
				SafeStatus:=3;
			END_IF
		END_IF
	3:
		IF fb_ton2.Q THEN
			IF Estop_RunAndRestart THEN
				Estop_RunAndRestart:=FALSE;
				fb_ton3.IN:=TRUE;
				SafeStatus:=4;
			END_IF
		END_IF
	4:
		IF fb_ton3.Q THEN
			IF Estop_Out THEN
				SafePLCRunOK:=TRUE;
				SafeStatus:=0;
			ELSE
				SafePLCRunOK:=FALSE;
				//Error:=TRUE;
				//ErrorId:=301;
				//ErrorDescription:='SafePLCRunOK fail';
			END_IF
		fb_ton0.IN:=FALSE;
		fb_ton1.IN:=FALSE;
		fb_ton2.IN:=FALSE;
		fb_ton3.IN:=FALSE;
		END_IF


END_CASE
END_ACTION

ACTION A_SetAxisPosition:
fb_ton4(PT:=t#0.5s);
CASE SetAxisPosState OF
	0:	(*FB_Set_AxisPosition*)
		FB_Set_AxisPosition(Execute:=TRUE);
		fb_ton4.IN:=TRUE;
		SetAxisPosState:=1;
	1:	(*wait*)
		FB_Set_AxisPosition();
		IF NOT FB_Set_AxisPosition.Done THEN		(*FB_Set_AxisPositionÃ»ÓÐÖ´ÐÐÍê£¬wait£¬³¬Ê±FB Error*)
			IF NOT fb_ton4.Q THEN
				SetAxisPosState:=1;
			ELSE
				SetAxisPosState:=99;
			END_IF
		ELSE
			SetAxisPosState:=88;
		END_IF
	88:
		SetAxisPosState:=0;
		SetAxisPositionDone:=TRUE;
		Error:=FALSE;
		ErrorID:=0;
		FB_Set_AxisPosition.Execute:=FALSE;
		fb_ton4.IN:=FALSE;
	99:
		SetAxisPosState:=99;
		SetAxisPositionDone:=FALSE;
		Error:=TRUE;
		FB_Set_AxisPosition.Execute:=FALSE;
		fb_ton4.IN:=FALSE;
		LED_Error:=TRUE;
		ErrorID:=401;
		ErrorDescription:='SetAxisPosition fail';
END_CASE
END_ACTION

ACTION A_SetLinearEncoderPositionBias:
//设置bias开始
A_SetLinearEncoderPositionBiasMC();
PositionBiasTON(PT:=T#0.1S);
CASE state_setLEPosBias OF
	0:
		PositionBiasTON.IN:=TRUE;
		IF MC_SetLEPosBias_PhaseShifter.Error THEN
			state_setLEPosBias:=-100;
		ELSE 
			state_setLEPosBias:=1;
		END_IF
	1:
		IF NOT MC_SetLEPosBias_PhaseShifter.Done  THEN
			MC_SetLEPosBias_PhaseShifter.Execute:=TRUE;
			state_setLEPosBias:=2;
		ELSE
			state_setLEPosBias:=-100;
		END_IF
	2:
		IF NOT MC_SetLEPosBias_PhaseShifter.Done THEN
			IF NOT PositionBiasTON.Q THEN
				state_setLEPosBias:=2;
			ELSE
				state_setLEPosBias:=-100;
			END_IF
		END_IF
		IF  MC_SetLEPosBias_PhaseShifter.Done THEN
			state_setLEPosBias:=88;
		END_IF	
		IF MC_SetLEPosBias_PhaseShifter.Error THEN
			state_setLEPosBias:=-100;
		END_IF 
		
	88:
		PositionBiasTON.IN:=FALSE;
		PositionBiasDone:=TRUE;
	-100:
		PositionBiasTON.IN:=FALSE;
		PositionBiasDone:=FALSE;
		Error:=TRUE;
		ErrorId:=901;
		ErrorDescription:='Set LinearEncoderPositionBias Error';
		Plc_EmergencyStop:=FALSE;
END_CASE
END_ACTION

ACTION A_SetLinearEncoderPositionBiasMC:
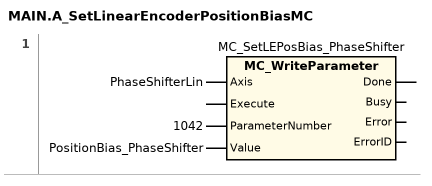
// NETWORK 1
MC_SetLEPosBias_PhaseShifter(
    Axis := PhaseShifterLin,
    ParameterNumber := 1042,
    Value := PositionBias_PhaseShifter); // MC_WriteParameter
END_ACTION

ACTION A_SetMotorAxisPosition:
fb_ton4_2(PT:=T#0.5S);
CASE SetMotorAxisPosState OF
	0:	(*FB_Set_AxisPosition*)
		FB_Set_MotorAxisPosition(Execute:=TRUE);
		fb_ton4_2.IN:=TRUE;
		SetMotorAxisPosState:=1;
	1:	(*wait*)
		FB_Set_MotorAxisPosition();
		IF NOT FB_Set_MotorAxisPosition.Done THEN		
			IF NOT fb_ton4_2.Q THEN
				SetMotorAxisPosState:=1;
			ELSE
				SetMotorAxisPosState:=99;
			END_IF
		ELSE
			SetMotorAxisPosState:=88;
		END_IF
	88:
		SetMotorAxisPosState:=0;
		SetMotorAxisPositionDone:=TRUE;
		Error:=FALSE;
		ErrorID:=0;
		FB_Set_MotorAxisPosition.Execute:=FALSE;
		fb_ton4_2.IN:=FALSE;
	99:
		SetMotorAxisPosState:=99;
		SetMotorAxisPositionDone:=FALSE;
		Error:=TRUE;
		FB_Set_MotorAxisPosition.Execute:=FALSE;
		fb_ton4.IN:=FALSE;
		LED_Error:=TRUE;
		ErrorID:=401;
		ErrorDescription:='SetMotorAxisPosition fail';
END_CASE
END_ACTION

END_PROGRAM

(* stored: Version 1.1.0.1, ProductVersion 3.1.4024.6
   POU MAIN: Id {9221b602-3f7e-4757-b581-54b56182ad8f}, SpecialFunc None
   Folder Axis: Id {1f5db9b2-f074-43bd-a7a5-f28b002c6ac6}
   Folder Check: Id {79c48f21-8e44-4159-8773-87594d6e7620}
   Folder Driver: Id {06d9eaf4-b0e1-444b-9d9d-89e6e18ffc32}
   Folder LinearEncoder: Id {4f24c8b2-fa71-4a79-b365-8e83326d2610}
   Folder Recipe: Id {c556f121-0220-445e-afd2-6e585e1080be}
   Folder Safe: Id {8d52a6a5-8a59-474d-a357-67246f4286de}
   Folder TC: Id {4ef3e57e-ed4b-4379-8b8b-cf198d1ecdc5}
   Action A_CheckHardwareEmergencyStopStatus: Id {c59a955b-0a8f-43a7-a0e7-3ab11b3d5ab6}
   Action A_CheckKillSwitch: Id {158eed83-fba1-4051-b569-3585448d2a5a}
   Action A_CheckLimitSwitch: Id {1026ae85-58e3-4004-8dd3-becfab0085f9}
   Action A_CheckLinearEncoder: Id {04ef6a41-e2ba-498d-aa00-f823237bb5de}
   Action A_CheckMaxVelocity: Id {b95fb694-2a75-4423-bee6-d704fd7332fe}
   Action A_GetDriverStatus: Id {e05cf975-7b3e-4430-bb2e-a308f4391f1b}
   Action A_GetDriverStatusMC: Id {2d8972a4-2924-4445-a68a-757b585b0760}
   Action A_GetMotorTemperature: Id {177f6aa7-fb59-4f66-a7a6-1b4260347e60}
   Action A_InitAxisParameters: Id {a92c2dd6-12b0-4a71-a4bc-d7afbc965cb4}
   Action A_InitRecipeParameters: Id {6aa76980-7ae7-46e7-9688-f94b6fa6510d}
   Action A_KillOpcIocShellExe: Id {e0252576-ad9e-49ed-bcc5-7f64aacd5ffe}
   Action A_LEHeartBeatMonitor: Id {c15e81d3-3944-4229-9ecc-53c2921ba7f3}
   Action A_LoadOpcIocShellExe: Id {e69e9ea4-205f-45b3-85e7-e1c1b3150dfb}
   Action A_MonitorMotorAndLE: Id {8906040e-6c25-4137-b340-4fb081d521ce}
   Action A_PosDiffDetectiion: Id {e857c546-d367-4f19-9434-ed29c144eb6f}
   Action A_RestartDrivers: Id {d1732994-27d5-4d0a-bd2e-fb077b65c9a9}
   Action A_RestartTC: Id {737d9420-c364-46ec-805e-ce283c214994}
   Action A_SafePlcStartInit: Id {4d1a8480-9923-4117-8ca7-ea613a82dfad}
   Action A_SetAxisPosition: Id {eb32aedd-8f01-44b1-96a9-73f233ea8548}
   Action A_SetLinearEncoderPositionBias: Id {6f3d3f8e-255d-4e09-853f-5fdf91122229}
   Action A_SetLinearEncoderPositionBiasMC: Id {d950edd3-252b-4c3c-9e26-a84e2707fa62}
   Action A_SetMotorAxisPosition: Id {1f7b7b3c-5e38-4a99-82a4-a1df4bf05d0c} *)
